{attribute 'linkalways'}
{attribute 'no_explicit_call' := 'This FB is a CLASS and must be accessed using methods or properties'}
{attribute 'enable_dynamic_creation'}
FUNCTION_BLOCK Node_F_VN_RemapImageToLogPolarSpaceExp2 EXTENDS VisionNode
VAR
    ipSrcImage : _ITcVnImage;
    ipDestImage : _ITcVnImage;
    aCenter : _TcVnPoint2_REAL;
    fScale : _LREAL(0);
    eInterpolationType : _ETcVnInterpolationType(ETcVnInterpolationType.TCVN_IT_BILINEAR);
    nDestWidth : _DINT(-1);
    nDestHeight : _DINT(-1);
    hrPrev : _HRESULT(S_OK);
    hresult : _HRESULT(S_OK);
END_VAR

METHOD PUBLIC Clone : I_Node
VAR
    pNode : POINTER TO Node_F_VN_RemapImageToLogPolarSpaceExp2;
END_VAR
pNode := __NEW(Node_F_VN_RemapImageToLogPolarSpaceExp2);
Clone := pNode^;
END_METHOD

METHOD FB_init : BOOL
VAR_INPUT
    bInitRetains : BOOL;
    bInCopyCode : BOOL;
END_VAR
AddInput('ipSrcImage', ipSrcImage);
AddOutput('ipDestImage', ipDestImage);
AddInput('aCenter', aCenter);
AddParameter('fScale', fScale);
AddParameter('eInterpolationType', eInterpolationType);
AddParameter('nDestWidth', nDestWidth);
AddParameter('nDestHeight', nDestHeight);
AddInput('hrPrev', hrPrev);
AddOutput('hresult', hresult);
END_METHOD

METHOD PROTECTED OnExecute
hresult.Value := F_VN_RemapImageToLogPolarSpaceExp2(
    ipSrcImage := ipSrcImage.Value,
    ipDestImage := ipDestImage.Value,
    aCenter := aCenter.Value,
    fScale := fScale.Value,
    eInterpolationType := eInterpolationType.Value,
    nDestWidth := nDestWidth.Value,
    nDestHeight := nDestHeight.Value,
    hrPrev := hrPrev.Value);
END_METHOD

METHOD PUBLIC PreExecutionCheck
VAR_INPUT
    Check : I_PreExecutionChecks;
END_VAR
Check.IsTrue(ipSrcImage.IsValid, 'ipSrcImage must contain an image');
Check.IsTrue((ipDestImage.Value = 0) OR (ipDestImage.Value <> ipSrcImage.Value), 'Destination must be different from the source image');
Check.IsTrue((eInterpolationType.Value = ETcVnInterpolationType.TCVN_IT_NEAREST_NEIGHBOR) OR
             (eInterpolationType.Value = ETcVnInterpolationType.TCVN_IT_BILINEAR) OR
             (eInterpolationType.Value = ETcVnInterpolationType.TCVN_IT_BICUBIC) OR
             (eInterpolationType.Value = ETcVnInterpolationType.TCVN_IT_AREA_BASED) OR
             (eInterpolationType.Value = ETcVnInterpolationType.TCVN_IT_LANCZOS4), 'Unsupported eInterpolationType');
Check.IsTrue(nDestWidth.Value >= -1, 'Destination width must be -1 for source width, 0 for automatic, or positive');
Check.IsTrue(nDestHeight.Value >= -1, 'Destination height must be -1 for source height, 0 for automatic, or positive');
END_METHOD

END_FUNCTION_BLOCK

(* stored: Version 1.1.0.1, ProductVersion 3.1.4026.19
   POU Node_F_VN_RemapImageToLogPolarSpaceExp2: Id {ab55bf34-8973-4897-b7ed-3b9760cc4ded}, SpecialFunc None
   Folder Constructor: Id {087f6471-b9be-4310-b1b7-8c91ec0a432c}
   Method Clone: Id {17c5af51-314d-4790-a0bc-b25e755e7a00}
   Method FB_init: Id {8ce76426-19eb-4bab-9285-80c34a607cb0}
   Method OnExecute: Id {1c3785f9-69c7-4b42-930e-0a8adda3bee9}
   Method PreExecutionCheck: Id {51309e9d-a3b3-46a3-b51e-c63ad9f1497d} *)
